FUNCTION_BLOCK CmdSludgeDischargeSLB (* CAT Function Block Type *)
  (* Standard: 61499-2 *)
  (* Version 2.0, 10/1/2026, Claude/Hidryco, Schneider Electric, Rev2 - Cmin (velocidade minima por bomba) do IThis para a logica; Rev1 - Nivel L (49LT0001) e parametros de pausa T_Restart/T_FlowLL (persistentes) *)
  PACKAGE SE.Nereda;
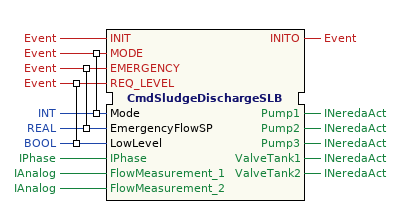
  EVENT_INPUT
    INIT;
    MODE WITH Mode;
    EMERGENCY WITH EmergencyFlowSP;
    REQ_LEVEL WITH LowLevel; (* Nivel L do 49LT0001 *)
  END_EVENT
  EVENT_OUTPUT
    INITO;
  END_EVENT
  VAR_INPUT
    Mode : INT;
    EmergencyFlowSP : REAL;
    LowLevel : BOOL; (* Nivel L do 49LT0001 (pausa a descarga) *)
  END_VAR
  SOCKETS
    IPhase : IPhase;
  END_SOCKETS
  SOCKETS
    FlowMeasurement_1 : IAnalog;
    FlowMeasurement_2 : IAnalog;
  END_SOCKETS
  PLUGS
    Pump1 : INeredaAct;
    Pump2 : INeredaAct;
    Pump3 : INeredaAct;
    ValveTank1 : INeredaAct;
    ValveTank2 : INeredaAct;
  END_PLUGS
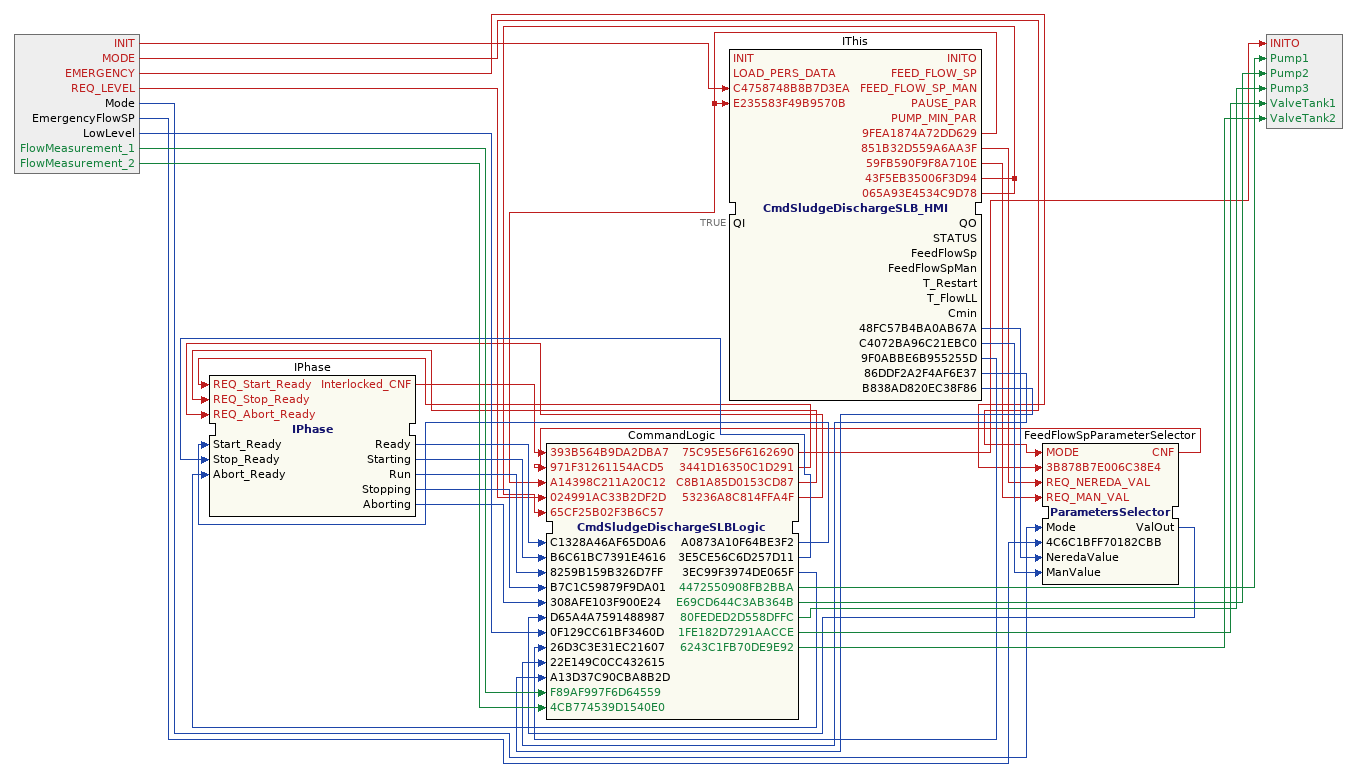
  (* 01 - FUNCTIONNAL INPUT INTERFACE *)
  (* 00 - INITIALIZATION *)
  (* 05 - LOGIC *)
  (* 06 - HMI INTERFACE *)
  (* 03 - FIELD INTERFACE *)
  (* 02 - FUNCTIONNAL OUTPUT INTERFACE *)
  (* Command Logic *)
  (* Capacity Setpoint *)
  FBS
    IThis : CmdSludgeDischargeSLB_HMI(QI := TRUE);
    FeedFlowSpParameterSelector : ParametersSelector;
    CommandLogic : CmdSludgeDischargeSLBLogic;
  END_FBS
  EVENT_CONNECTIONS
    MODE TO FeedFlowSpParameterSelector.MODE;
    EMERGENCY TO FeedFlowSpParameterSelector.3B878B7E006C38E4;
    IPhase.Interlocked_CNF TO CommandLogic.393B564B9DA2DBA7;
    FeedFlowSpParameterSelector.CNF TO CommandLogic.971F31261154ACD5;
    INIT TO IThis.C4758748B8B7D3EA;
    IThis.9FEA1874A72DD629 TO CommandLogic.A14398C211A20C12;
    IThis.851B32D559A6AA3F TO FeedFlowSpParameterSelector.REQ_NEREDA_VAL;
    IThis.59FB590F9F8A710E TO FeedFlowSpParameterSelector.REQ_MAN_VAL;
    CommandLogic.75C95E56F6162690 TO INITO;
    IThis.9FEA1874A72DD629 TO IThis.E235583F49B9570B;
    CommandLogic.3441D16350C1D291 TO IPhase.REQ_Start_Ready;
    CommandLogic.C8B1A85D0153CD87 TO IPhase.REQ_Stop_Ready;
    CommandLogic.53236A8C814FFA4F TO IPhase.REQ_Abort_Ready;
    REQ_LEVEL TO CommandLogic.024991AC33B2DF2D;
    IThis.43F5EB35006F3D94 TO CommandLogic.65CF25B02F3B6C57;
    IThis.065A93E4534C9D78 TO CommandLogic.65CF25B02F3B6C57;
  END_CONNECTIONS
  DATA_CONNECTIONS
    Mode TO FeedFlowSpParameterSelector.Mode;
    EmergencyFlowSP TO FeedFlowSpParameterSelector.4C6C1BFF70182CBB;
    IPhase.Ready TO CommandLogic.C1328A46AF65D0A6;
    IPhase.Starting TO CommandLogic.B6C61BC7391E4616;
    IPhase.Run TO CommandLogic.8259B159B326D7FF;
    IPhase.Stopping TO CommandLogic.B7C1C59879F9DA01;
    IPhase.Aborting TO CommandLogic.308AFE103F900E24;
    FeedFlowSpParameterSelector.ValOut TO CommandLogic.D65A4A7591488987;
    IThis.48FC57B4BA0AB67A TO FeedFlowSpParameterSelector.NeredaValue;
    IThis.C4072BA96C21EBC0 TO FeedFlowSpParameterSelector.ManValue;
    CommandLogic.A0873A10F64BE3F2 TO IPhase.Start_Ready;
    CommandLogic.3E5CE56C6D257D11 TO IPhase.Stop_Ready;
    CommandLogic.3EC99F3974DE065F TO IPhase.Abort_Ready;
    LowLevel TO CommandLogic.0F129CC61BF3460D;
    IThis.9F0ABBE6B955255D TO CommandLogic.26D3C3E31EC21607;
    IThis.86DDF2A2F4AF6E37 TO CommandLogic.22E149C0CC432615;
    IThis.B838AD820EC38F86 TO CommandLogic.A13D37C90CBA8B2D;
  END_CONNECTIONS
  ADAPTER_CONNECTIONS
    CommandLogic.4472550908FB2BBA TO Pump1;
    CommandLogic.E69CD644C3AB364B TO Pump2;
    CommandLogic.80FEDED2D558DFFC TO Pump3;
    CommandLogic.1FE182D7291AACCE TO ValveTank1;
    CommandLogic.6243C1FB70DE9E92 TO ValveTank2;
    FlowMeasurement_1 TO CommandLogic.F89AF997F6D64559;
    FlowMeasurement_2 TO CommandLogic.4CB774539D1540E0;
  END_CONNECTIONS
END_FUNCTION_BLOCK
